{attribute 'GeneratedUsingTerminal: EL9540-0010-0016'}
{attribute addProperty BoxType "EL9540-0010-0016"}
{attribute addProperty Id "EtcSlaveTerminalBaseStatus_UpAT %I*Status_Up_DB3531282WcStateAT %I*WcState_9091E0EB2InfoDataAT %I*InfoData_6F19DB2B2"}
{attribute addProperty CRC "3483813640"}
{attribute addProperty Size "6"}
TYPE EL9540_CFA6C708 EXTENDS EtcSlaveTerminalBase :
STRUCT
	{attribute addProperty Name "Status_Up"}
	Status_Up : Status_Up_DB353128;
	{attribute addProperty Name "WcState"}
	WcState : WcState_9091E0EB;
	{attribute addProperty Name "InfoData"}
	InfoData : InfoData_6F19DB2B;
END_STRUCT
END_TYPE

(* stored: Version 1.2.0.0, ProductVersion 3.1.4024.9
   DUT EL9540_CFA6C708: Id {7a226f44-fc27-481e-8a14-2b21b5258df4} *)
